// Mitsubishi GX Works2 project: 24   PLC: FX3G

// task Task_01 (event TRUE, interval 0, priority 31): POU_01

PROGRAM POU_01
VAR
  wstep : INT;
  counter : INT;
  ton1 : TON;
END_VAR
M99 := FALSE AND
M1 AND M2 AND
Y0 AND Y1 AND Y2 AND Y3;

IF M8002 THEN
	wstep := 0;
END_IF;

CASE wstep OF
	0:
		zrst(TRUE, Y0, Y3);
		ton1(in := FALSE);
		counter := 0;
		
		IF M1 THEN	
			wstep := 20;
		END_IF;
		
	20:
		zrst(TRUE, Y0, Y2);
		Z0 := counter;
		Y0Z0 := TRUE;
		
		ton1(in := NOT ton1.q, pt := t#0.5s);
		IF ton1.q THEN
			counter := counter + 1;
			counter := counter MOD 3;
		END_IF;
		
		IF M2 THEN
			wstep := 21;
		END_IF;
	21:
		zrst(TRUE, Y0, Y2);
		Y3 := TRUE;
		ton1(in := NOT ton1.q, pt := t#5s);
		
		IF ton1.q THEN
			wstep := 0;
		END_IF;
END_CASE;
END_PROGRAM
